FUNCTION_BLOCK EVENT_CONTROLLER (* Composite Function Block Type *)
  (* Standard: 61499-2 *)
  (* Version 1.0, 2019-03-16, adeel *)
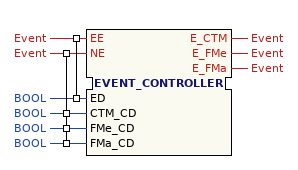
  EVENT_INPUT
    EE WITH ED;
    NE WITH CTM_CD, FMe_CD, FMa_CD;
  END_EVENT
  EVENT_OUTPUT
    E_CTM; (* Execution Confirmation *)
    E_FMe;
    E_FMa;
  END_EVENT
  VAR_INPUT
    ED : BOOL;
    CTM_CD : BOOL; (* Input event qualifier *)
    FMe_CD : BOOL;
    FMa_CD : BOOL;
  END_VAR
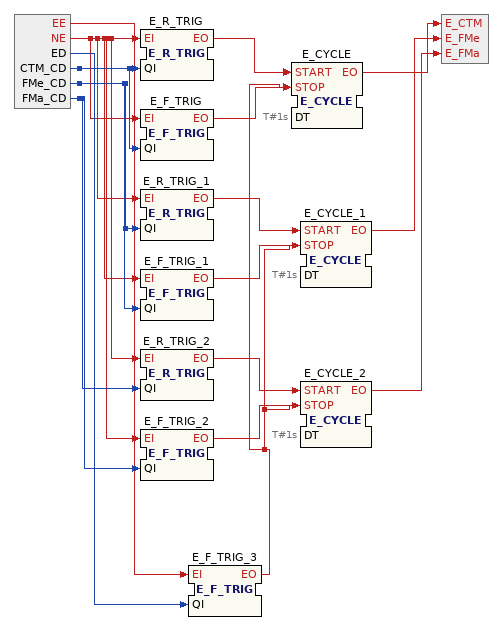
  FBS
    E_F_TRIG : E_F_TRIG;
    E_R_TRIG : E_R_TRIG;
    E_CYCLE : E_CYCLE(DT := T#1s);
    E_R_TRIG_1 : E_R_TRIG;
    E_F_TRIG_1 : E_F_TRIG;
    E_CYCLE_1 : E_CYCLE(DT := T#1s);
    E_R_TRIG_2 : E_R_TRIG;
    E_F_TRIG_2 : E_F_TRIG;
    E_CYCLE_2 : E_CYCLE(DT := T#1s);
    E_F_TRIG_3 : E_F_TRIG;
  END_FBS
  EVENT_CONNECTIONS
    E_R_TRIG.EO TO E_CYCLE.START;
    E_F_TRIG.EO TO E_CYCLE.STOP;
    E_CYCLE.EO TO E_CTM;
    NE TO E_F_TRIG_2.EI;
    E_CYCLE_1.EO TO E_FMe;
    E_CYCLE_2.EO TO E_FMa;
    E_R_TRIG_1.EO TO E_CYCLE_1.START;
    E_F_TRIG_1.EO TO E_CYCLE_1.STOP;
    E_R_TRIG_2.EO TO E_CYCLE_2.START;
    E_F_TRIG_2.EO TO E_CYCLE_2.STOP;
    EE TO E_F_TRIG_3.EI;
    E_F_TRIG_3.EO TO E_CYCLE.STOP;
    E_F_TRIG_3.EO TO E_CYCLE_1.STOP;
    E_F_TRIG_3.EO TO E_CYCLE_2.STOP;
    NE TO E_R_TRIG.EI;
    NE TO E_F_TRIG.EI;
    NE TO E_R_TRIG_1.EI;
    NE TO E_F_TRIG_1.EI;
    NE TO E_R_TRIG_2.EI;
  END_CONNECTIONS
  DATA_CONNECTIONS
    CTM_CD TO E_R_TRIG.QI;
    FMe_CD TO E_R_TRIG_1.QI;
    FMa_CD TO E_R_TRIG_2.QI;
    ED TO E_F_TRIG_3.QI;
    CTM_CD TO E_F_TRIG.QI;
    FMe_CD TO E_F_TRIG_1.QI;
    FMa_CD TO E_F_TRIG_2.QI;
  END_CONNECTIONS
END_FUNCTION_BLOCK
